(* Logix 5000 project; controller NSH_PLC1 vendor 1 type 14 code 167 rev 32.11; software revision 32.02; part 3 of 12 *)
(* tags used below, declared in another part *)
   M10 : Motor;   // Vib.
   M10A : Motor;   // Asp.
   M10B : Motor;   // Asp.
   M11 : Motor;   // Ele.
   M12aA : Motor;   // Grav.Sep
   M12aB : Motor;   // Syntron
   M13aA : Motor;   // Grav.Sep
   M13aB : Motor;   // Syntron
   M14 : Motor;   // Vib.
   M15 : Motor;   // Ele.
   M1A : Motor;   // Vib.
   M2 : Motor;   // Vib.
   M25 : Motor;   // Accept Vib.
   M27 : Motor;   // Belt
   M28 : Motor;   // Belt
   M29 : Motor;   // Ele.
   M3 : Motor;   // Belt
   M30A : Motor;   // HC Vib.
   M30B : Motor;   // Hard Crkr.
   M30C : Motor;   // Shr.Roll.
   M30D : Motor;   // Shr.Roll.
   M31A : Motor;   // Asp.
   M31B : Motor;   // Asp.
   M32A : Motor;   // Vib.Scrn.
   M32B : Motor;   // Ele.
   M33 : Motor;   // Belt
   M34 : Motor;   // Destoner
   M35 : Motor;   // Ele.
   M36A : Motor;   // G. Sep.
   M36B : Motor;   // R. Feeder.
   M37 : Motor;   // 5x12
   M38A : Motor;   // Asp.
   M38B : Motor;   // Asp.
   M39 : Motor;   // Ele.
   M4 : Motor;   // Vib.
   M40A : Motor;   // Sep.
   M40B : Motor;   // Syn.Fer.
   M41 : Motor;   // Ele.
   M44A : Motor;   // Belt
   M44B : Motor;   // Belt
   M5 : Motor;   // Vib.
   M6 : Motor;   // Belt
   M7 : Motor;   // Ele.
   M8 : Motor;   // Shkr.
   M9A : Motor;   // Asp.
   M9B : Motor;   // Asp.
   S11 : Motor;   // Ele.
   S32A : Motor;   // HC Vib.
   S32B : Motor;   // Hard Crkr.
   S32C : Motor;   // Shr.Roll.
   S32D : Motor;   // S.Roll
   S33A : Motor;   // HC Vib.
   S33B : Motor;   // Hard Crkr.
   S33C : Motor;   // Shr.Roll.
   S33D : Motor;   // S.Roll
   S37A : Motor;   // HC Vib.
   S37B : Motor;   // Hard Crkr.
   S37C : Motor;   // Shr.Roll.
   S37D : Motor;   // S.Roll
   S40A : Motor;   // HC Vib.
   S40B : Motor;   // Hard Crkr.
   S40C : Motor;   // Shr.Roll.
   S40D : Motor;   // S.Roll
   S42A : Motor;   // HC Vib.
   S42B : Motor;   // Hard Crkr.
   S42C : Motor;   // S.Roll
   S42D : Motor;   // Shr.Roll.
   S46A : Motor;   // HC Vib.
   S46B : Motor;   // Hard Crkr.
   S46C : Motor;   // S.Roll
   S46D : Motor;   // Shr.Roll.
(* HullerSheller, continued *)

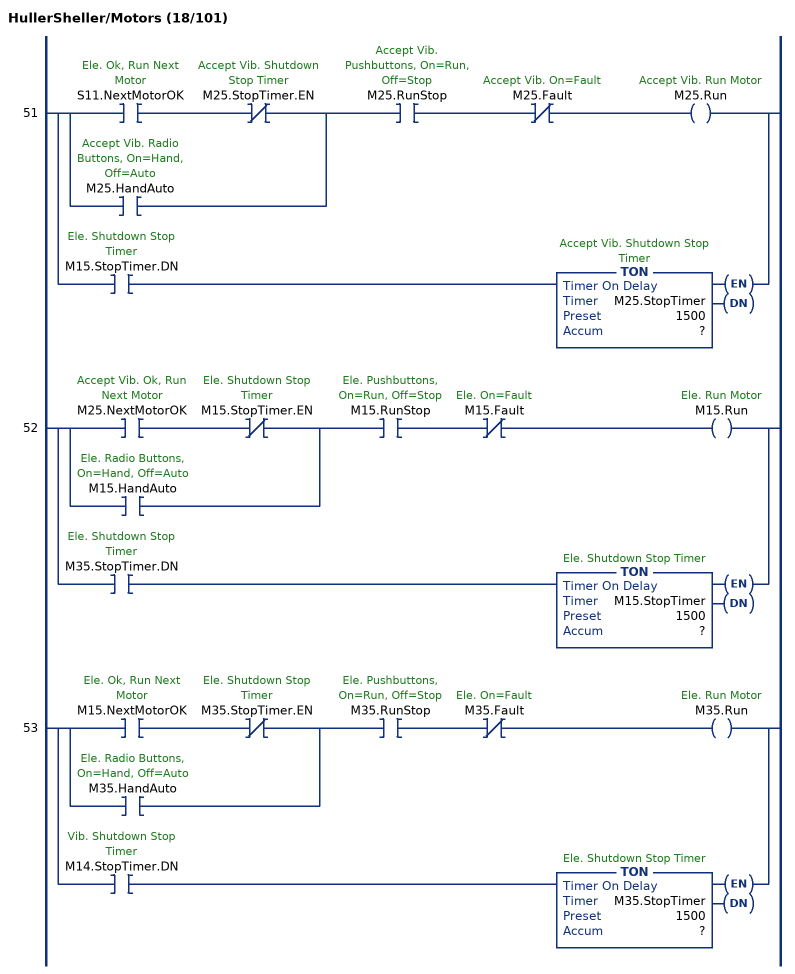
   [picture p42: HullerSheller/Motors rungs 51-53]
   51: [[XIC(S11.NextMotorOK) XIO(M25.StopTimer.EN) ,XIC(M25.HandAuto) ] XIC(M25.RunStop) XIO(M25.Fault) OTE(M25.Run) ,XIC(M15.StopTimer.DN) TON(M25.StopTimer,?,?) ];
   52: [[XIC(M25.NextMotorOK) XIO(M15.StopTimer.EN) ,XIC(M15.HandAuto) ] XIC(M15.RunStop) XIO(M15.Fault) OTE(M15.Run) ,XIC(M35.StopTimer.DN) TON(M15.StopTimer,?,?) ];
   53: [[XIC(M15.NextMotorOK) XIO(M35.StopTimer.EN) ,XIC(M35.HandAuto) ] XIC(M35.RunStop) XIO(M35.Fault) OTE(M35.Run) ,XIC(M14.StopTimer.DN) TON(M35.StopTimer,?,?) ];
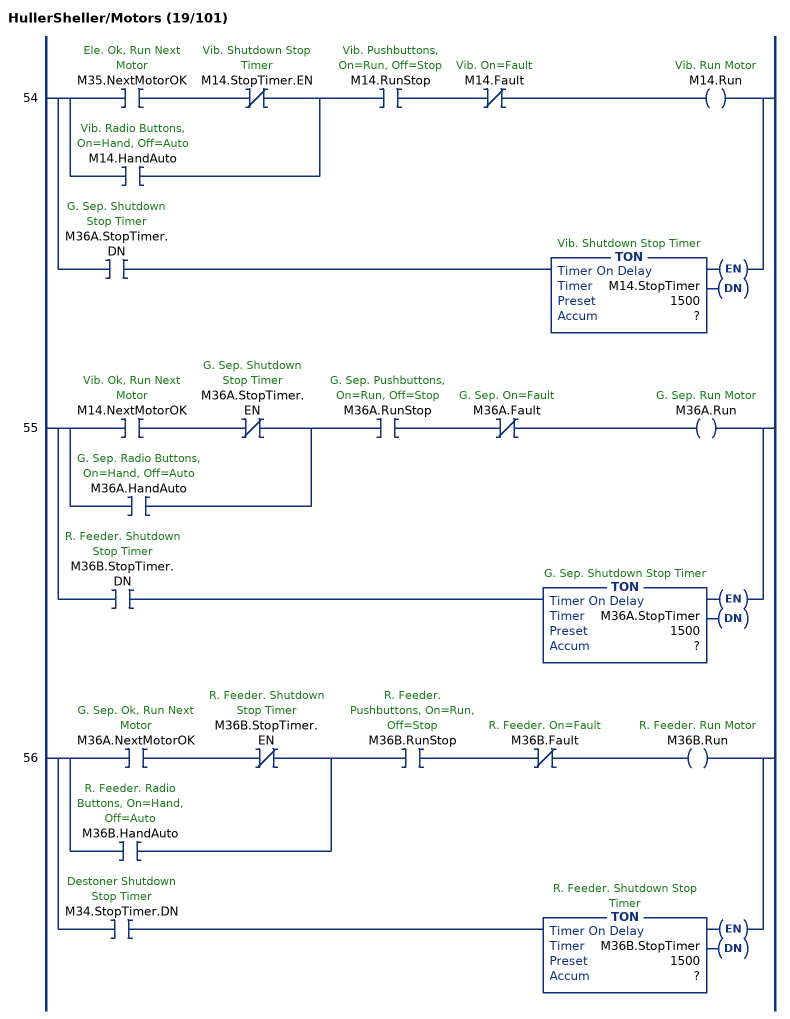
   54: [[XIC(M35.NextMotorOK) XIO(M14.StopTimer.EN) ,XIC(M14.HandAuto) ] XIC(M14.RunStop) XIO(M14.Fault) OTE(M14.Run) ,XIC(M36A.StopTimer.DN) TON(M14.StopTimer,?,?) ];
   55: [[XIC(M14.NextMotorOK) XIO(M36A.StopTimer.EN) ,XIC(M36A.HandAuto) ] XIC(M36A.RunStop) XIO(M36A.Fault) OTE(M36A.Run) ,XIC(M36B.StopTimer.DN) TON(M36A.StopTimer,?,?) ];
   56: [[XIC(M36A.NextMotorOK) XIO(M36B.StopTimer.EN) ,XIC(M36B.HandAuto) ] XIC(M36B.RunStop) XIO(M36B.Fault) OTE(M36B.Run) ,XIC(M34.StopTimer.DN) TON(M36B.StopTimer,?,?) ];
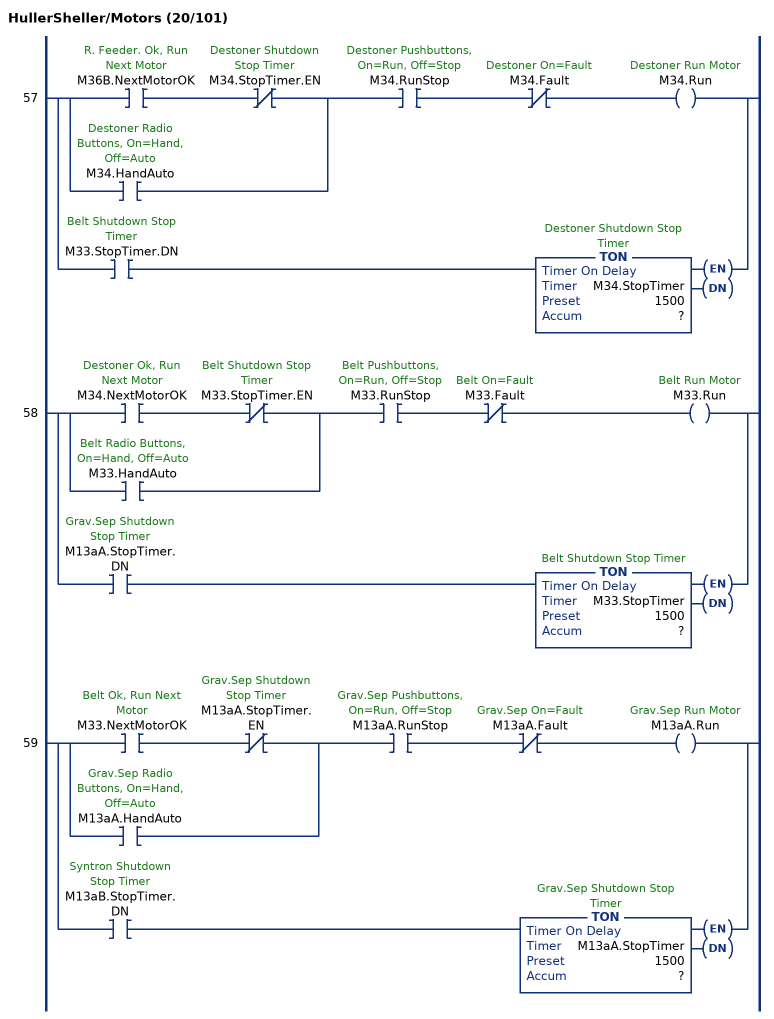
   57: [[XIC(M36B.NextMotorOK) XIO(M34.StopTimer.EN) ,XIC(M34.HandAuto) ] XIC(M34.RunStop) XIO(M34.Fault) OTE(M34.Run) ,XIC(M33.StopTimer.DN) TON(M34.StopTimer,?,?) ];
   58: [[XIC(M34.NextMotorOK) XIO(M33.StopTimer.EN) ,XIC(M33.HandAuto) ] XIC(M33.RunStop) XIO(M33.Fault) OTE(M33.Run) ,XIC(M13aA.StopTimer.DN) TON(M33.StopTimer,?,?) ];
   59: [[XIC(M33.NextMotorOK) XIO(M13aA.StopTimer.EN) ,XIC(M13aA.HandAuto) ] XIC(M13aA.RunStop) XIO(M13aA.Fault) OTE(M13aA.Run) ,XIC(M13aB.StopTimer.DN) TON(M13aA.StopTimer,?,?) ];
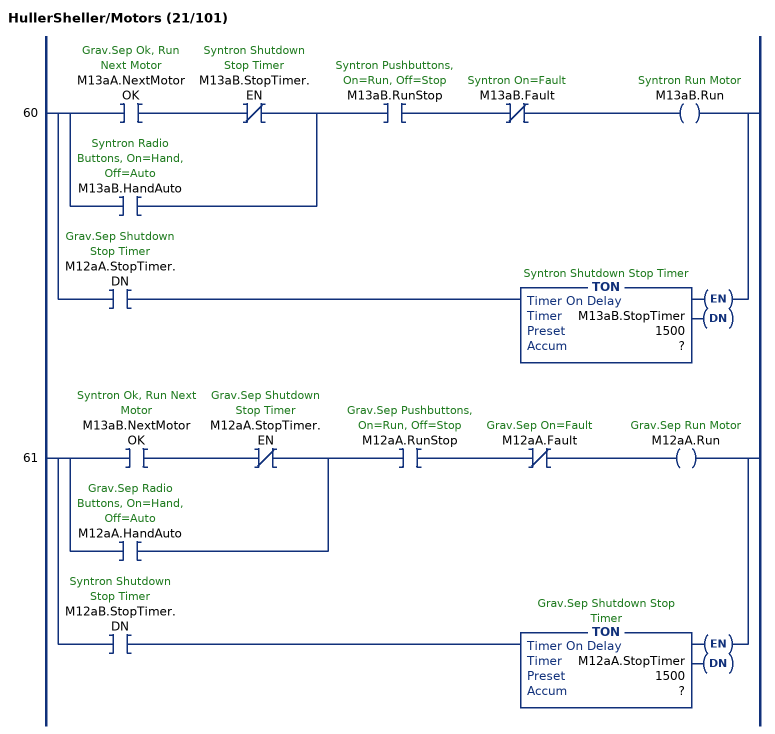
   60: [[XIC(M13aA.NextMotorOK) XIO(M13aB.StopTimer.EN) ,XIC(M13aB.HandAuto) ] XIC(M13aB.RunStop) XIO(M13aB.Fault) OTE(M13aB.Run) ,XIC(M12aA.StopTimer.DN) TON(M13aB.StopTimer,?,?) ];
   61: [[XIC(M13aB.NextMotorOK) XIO(M12aA.StopTimer.EN) ,XIC(M12aA.HandAuto) ] XIC(M12aA.RunStop) XIO(M12aA.Fault) OTE(M12aA.Run) ,XIC(M12aB.StopTimer.DN) TON(M12aA.StopTimer,?,?) ];
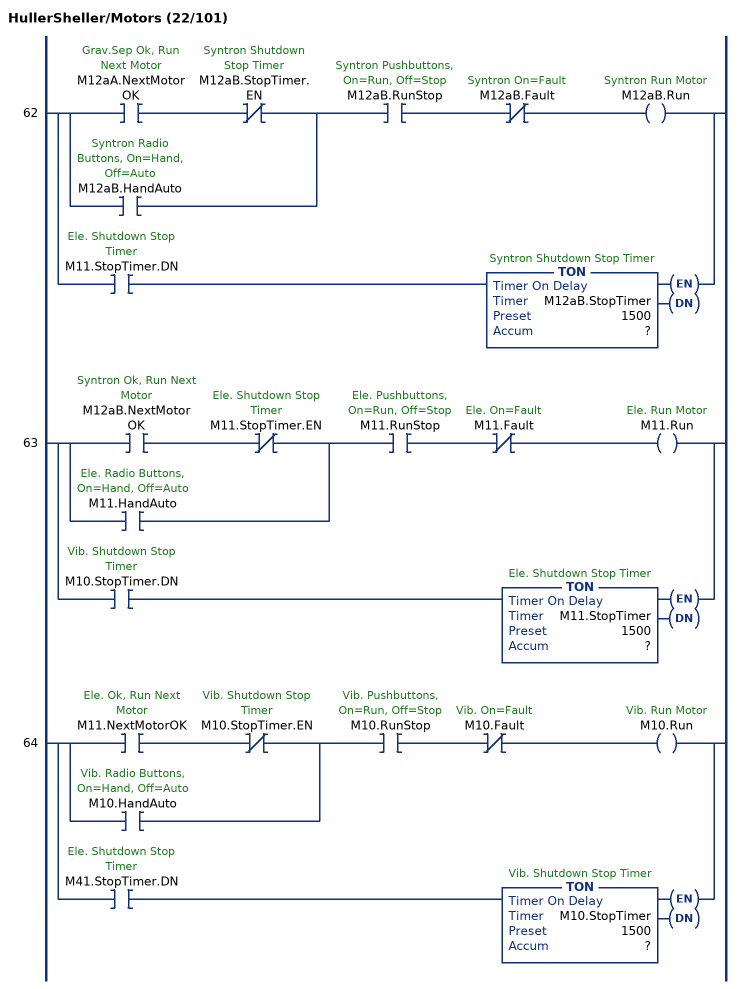
   62: [[XIC(M12aA.NextMotorOK) XIO(M12aB.StopTimer.EN) ,XIC(M12aB.HandAuto) ] XIC(M12aB.RunStop) XIO(M12aB.Fault) OTE(M12aB.Run) ,XIC(M11.StopTimer.DN) TON(M12aB.StopTimer,?,?) ];
   63: [[XIC(M12aB.NextMotorOK) XIO(M11.StopTimer.EN) ,XIC(M11.HandAuto) ] XIC(M11.RunStop) XIO(M11.Fault) OTE(M11.Run) ,XIC(M10.StopTimer.DN) TON(M11.StopTimer,?,?) ];
   64: [[XIC(M11.NextMotorOK) XIO(M10.StopTimer.EN) ,XIC(M10.HandAuto) ] XIC(M10.RunStop) XIO(M10.Fault) OTE(M10.Run) ,XIC(M41.StopTimer.DN) TON(M10.StopTimer,?,?) ];
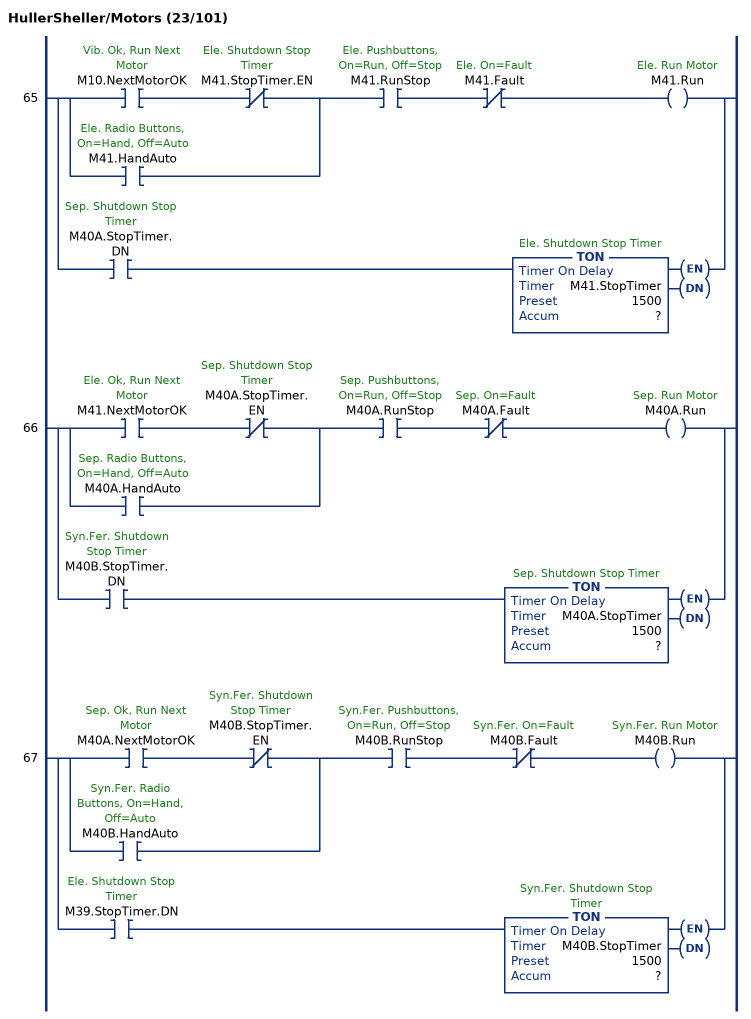
   65: [[XIC(M10.NextMotorOK) XIO(M41.StopTimer.EN) ,XIC(M41.HandAuto) ] XIC(M41.RunStop) XIO(M41.Fault) OTE(M41.Run) ,XIC(M40A.StopTimer.DN) TON(M41.StopTimer,?,?) ];
   66: [[XIC(M41.NextMotorOK) XIO(M40A.StopTimer.EN) ,XIC(M40A.HandAuto) ] XIC(M40A.RunStop) XIO(M40A.Fault) OTE(M40A.Run) ,XIC(M40B.StopTimer.DN) TON(M40A.StopTimer,?,?) ];
   67: [[XIC(M40A.NextMotorOK) XIO(M40B.StopTimer.EN) ,XIC(M40B.HandAuto) ] XIC(M40B.RunStop) XIO(M40B.Fault) OTE(M40B.Run) ,XIC(M39.StopTimer.DN) TON(M40B.StopTimer,?,?) ];
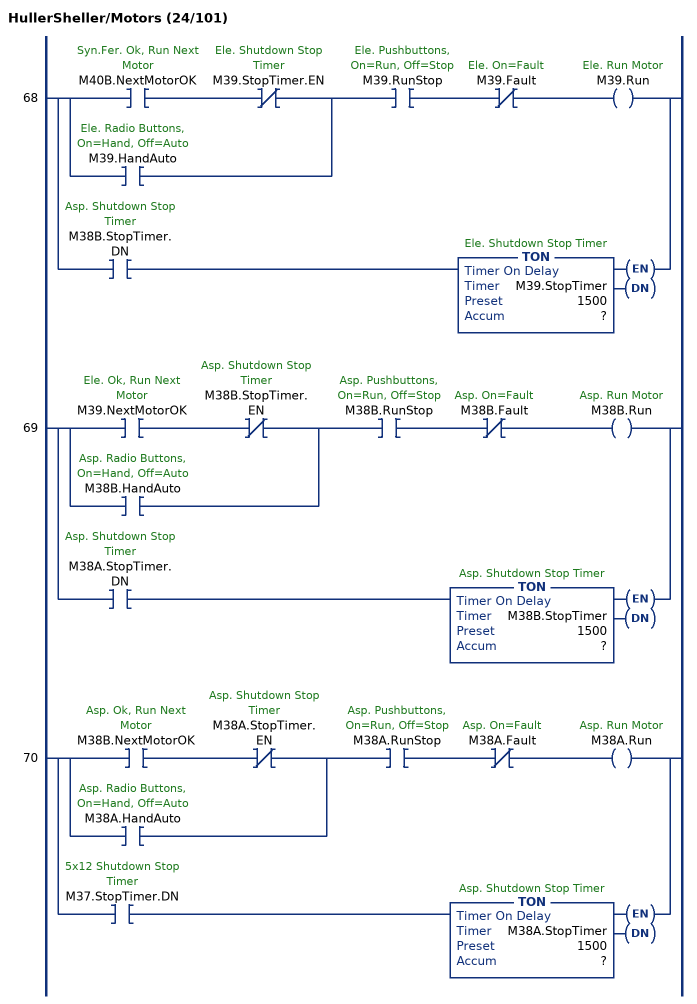
   68: [[XIC(M40B.NextMotorOK) XIO(M39.StopTimer.EN) ,XIC(M39.HandAuto) ] XIC(M39.RunStop) XIO(M39.Fault) OTE(M39.Run) ,XIC(M38B.StopTimer.DN) TON(M39.StopTimer,?,?) ];
   69: [[XIC(M39.NextMotorOK) XIO(M38B.StopTimer.EN) ,XIC(M38B.HandAuto) ] XIC(M38B.RunStop) XIO(M38B.Fault) OTE(M38B.Run) ,XIC(M38A.StopTimer.DN) TON(M38B.StopTimer,?,?) ];
   70: [[XIC(M38B.NextMotorOK) XIO(M38A.StopTimer.EN) ,XIC(M38A.HandAuto) ] XIC(M38A.RunStop) XIO(M38A.Fault) OTE(M38A.Run) ,XIC(M37.StopTimer.DN) TON(M38A.StopTimer,?,?) ];
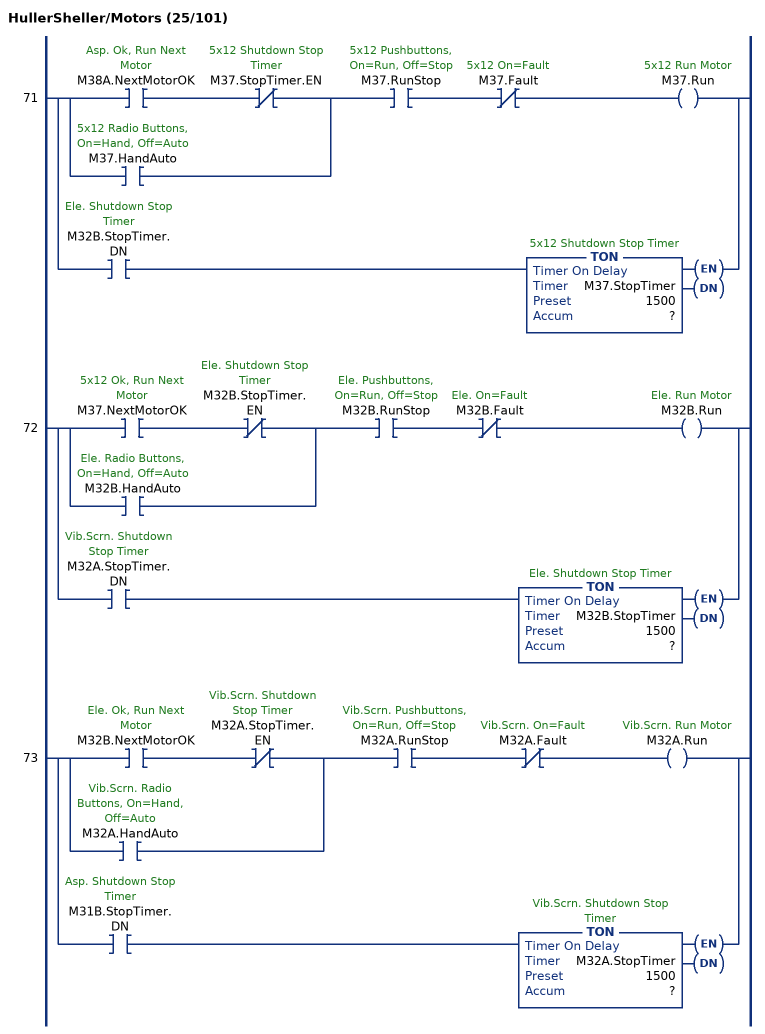
   71: [[XIC(M38A.NextMotorOK) XIO(M37.StopTimer.EN) ,XIC(M37.HandAuto) ] XIC(M37.RunStop) XIO(M37.Fault) OTE(M37.Run) ,XIC(M32B.StopTimer.DN) TON(M37.StopTimer,?,?) ];
   72: [[XIC(M37.NextMotorOK) XIO(M32B.StopTimer.EN) ,XIC(M32B.HandAuto) ] XIC(M32B.RunStop) XIO(M32B.Fault) OTE(M32B.Run) ,XIC(M32A.StopTimer.DN) TON(M32B.StopTimer,?,?) ];
   73: [[XIC(M32B.NextMotorOK) XIO(M32A.StopTimer.EN) ,XIC(M32A.HandAuto) ] XIC(M32A.RunStop) XIO(M32A.Fault) OTE(M32A.Run) ,XIC(M31B.StopTimer.DN) TON(M32A.StopTimer,?,?) ];
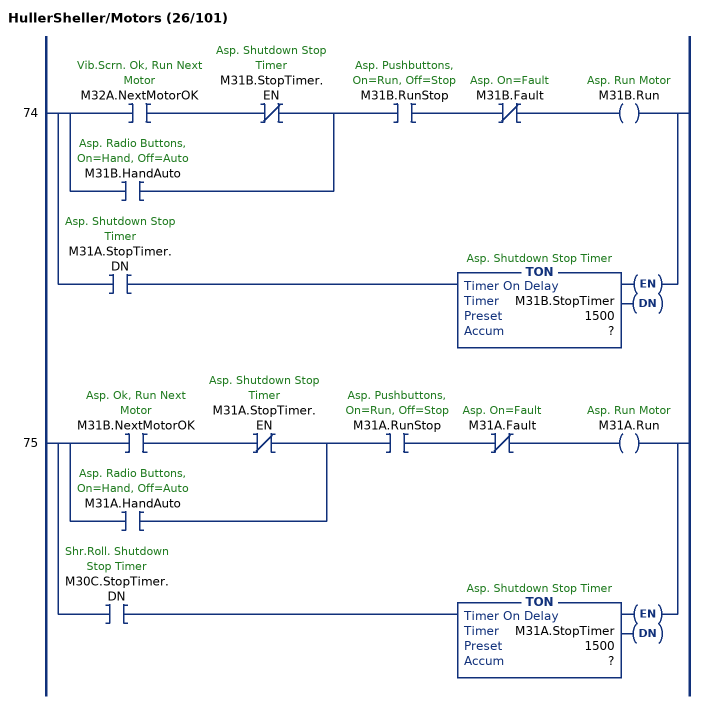
   74: [[XIC(M32A.NextMotorOK) XIO(M31B.StopTimer.EN) ,XIC(M31B.HandAuto) ] XIC(M31B.RunStop) XIO(M31B.Fault) OTE(M31B.Run) ,XIC(M31A.StopTimer.DN) TON(M31B.StopTimer,?,?) ];
   75: [[XIC(M31B.NextMotorOK) XIO(M31A.StopTimer.EN) ,XIC(M31A.HandAuto) ] XIC(M31A.RunStop) XIO(M31A.Fault) OTE(M31A.Run) ,XIC(M30C.StopTimer.DN) TON(M31A.StopTimer,?,?) ];
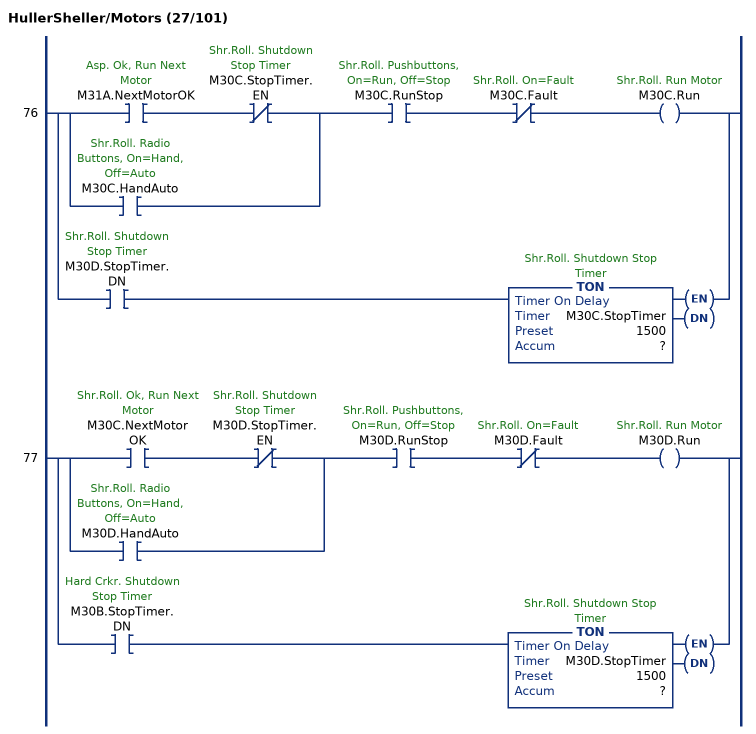
   76: [[XIC(M31A.NextMotorOK) XIO(M30C.StopTimer.EN) ,XIC(M30C.HandAuto) ] XIC(M30C.RunStop) XIO(M30C.Fault) OTE(M30C.Run) ,XIC(M30D.StopTimer.DN) TON(M30C.StopTimer,?,?) ];
   77: [[XIC(M30C.NextMotorOK) XIO(M30D.StopTimer.EN) ,XIC(M30D.HandAuto) ] XIC(M30D.RunStop) XIO(M30D.Fault) OTE(M30D.Run) ,XIC(M30B.StopTimer.DN) TON(M30D.StopTimer,?,?) ];
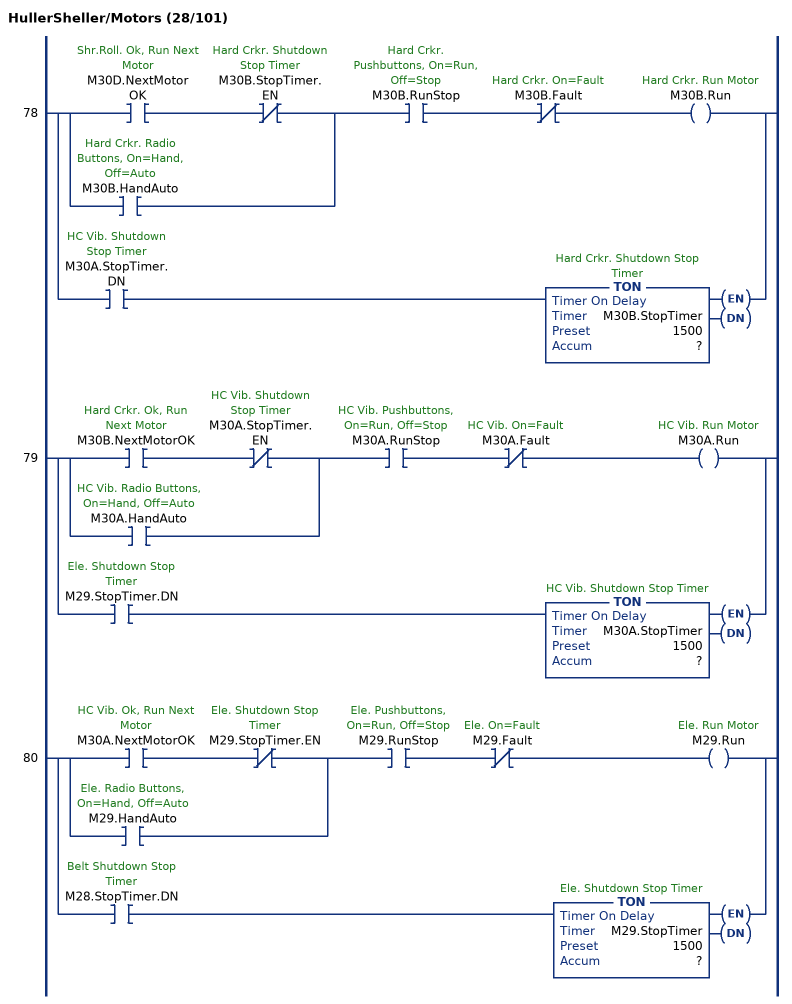
   78: [[XIC(M30D.NextMotorOK) XIO(M30B.StopTimer.EN) ,XIC(M30B.HandAuto) ] XIC(M30B.RunStop) XIO(M30B.Fault) OTE(M30B.Run) ,XIC(M30A.StopTimer.DN) TON(M30B.StopTimer,?,?) ];
   79: [[XIC(M30B.NextMotorOK) XIO(M30A.StopTimer.EN) ,XIC(M30A.HandAuto) ] XIC(M30A.RunStop) XIO(M30A.Fault) OTE(M30A.Run) ,XIC(M29.StopTimer.DN) TON(M30A.StopTimer,?,?) ];
   80: [[XIC(M30A.NextMotorOK) XIO(M29.StopTimer.EN) ,XIC(M29.HandAuto) ] XIC(M29.RunStop) XIO(M29.Fault) OTE(M29.Run) ,XIC(M28.StopTimer.DN) TON(M29.StopTimer,?,?) ];
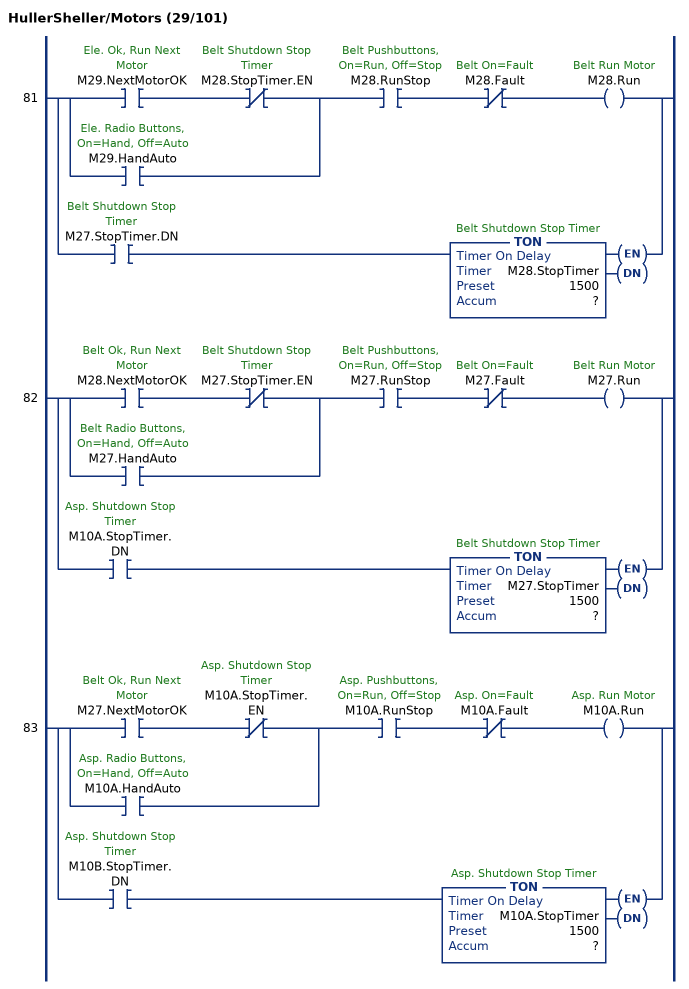
   81: [[XIC(M29.NextMotorOK) XIO(M28.StopTimer.EN) ,XIC(M29.HandAuto) ] XIC(M28.RunStop) XIO(M28.Fault) OTE(M28.Run) ,XIC(M27.StopTimer.DN) TON(M28.StopTimer,?,?) ];
   82: [[XIC(M28.NextMotorOK) XIO(M27.StopTimer.EN) ,XIC(M27.HandAuto) ] XIC(M27.RunStop) XIO(M27.Fault) OTE(M27.Run) ,XIC(M10A.StopTimer.DN) TON(M27.StopTimer,?,?) ];
   83: [[XIC(M27.NextMotorOK) XIO(M10A.StopTimer.EN) ,XIC(M10A.HandAuto) ] XIC(M10A.RunStop) XIO(M10A.Fault) OTE(M10A.Run) ,XIC(M10B.StopTimer.DN) TON(M10A.StopTimer,?,?) ];
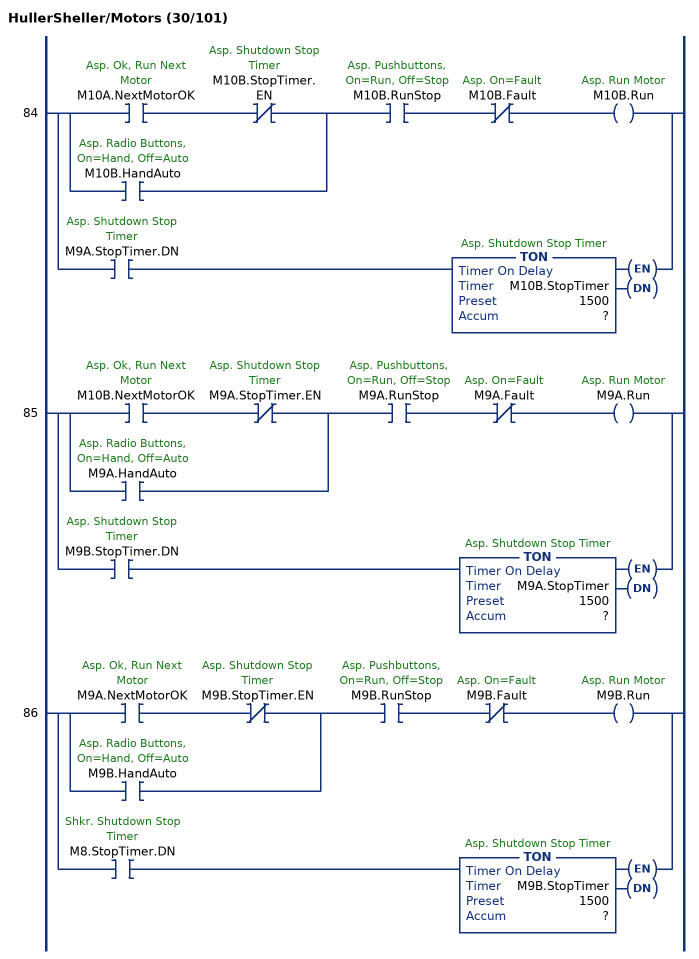
   84: [[XIC(M10A.NextMotorOK) XIO(M10B.StopTimer.EN) ,XIC(M10B.HandAuto) ] XIC(M10B.RunStop) XIO(M10B.Fault) OTE(M10B.Run) ,XIC(M9A.StopTimer.DN) TON(M10B.StopTimer,?,?) ];
   85: [[XIC(M10B.NextMotorOK) XIO(M9A.StopTimer.EN) ,XIC(M9A.HandAuto) ] XIC(M9A.RunStop) XIO(M9A.Fault) OTE(M9A.Run) ,XIC(M9B.StopTimer.DN) TON(M9A.StopTimer,?,?) ];
   86: [[XIC(M9A.NextMotorOK) XIO(M9B.StopTimer.EN) ,XIC(M9B.HandAuto) ] XIC(M9B.RunStop) XIO(M9B.Fault) OTE(M9B.Run) ,XIC(M8.StopTimer.DN) TON(M9B.StopTimer,?,?) ];
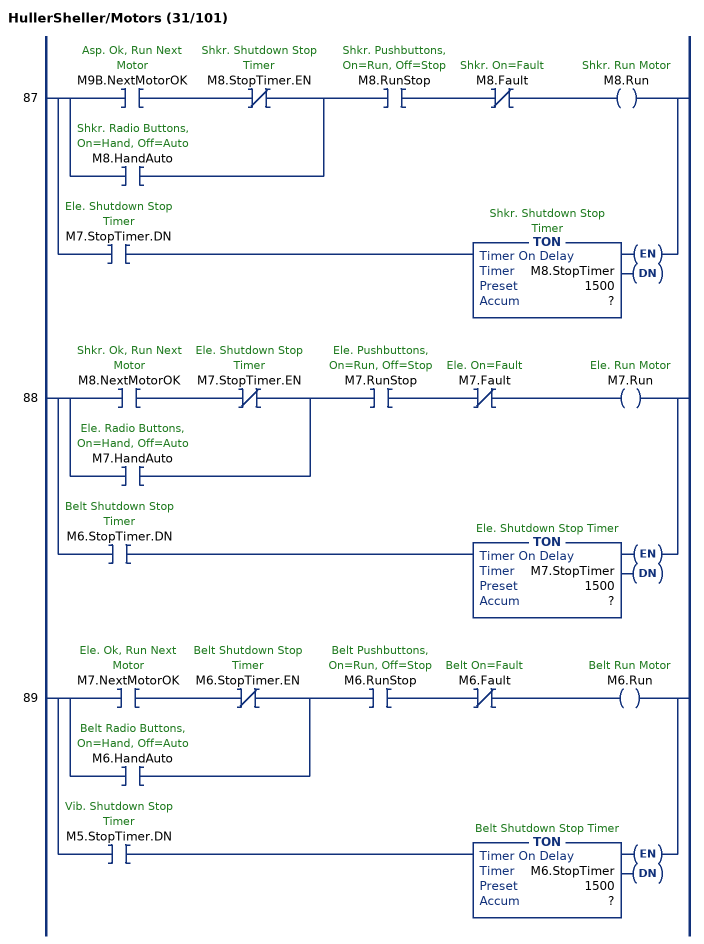
   87: [[XIC(M9B.NextMotorOK) XIO(M8.StopTimer.EN) ,XIC(M8.HandAuto) ] XIC(M8.RunStop) XIO(M8.Fault) OTE(M8.Run) ,XIC(M7.StopTimer.DN) TON(M8.StopTimer,?,?) ];
   88: [[XIC(M8.NextMotorOK) XIO(M7.StopTimer.EN) ,XIC(M7.HandAuto) ] XIC(M7.RunStop) XIO(M7.Fault) OTE(M7.Run) ,XIC(M6.StopTimer.DN) TON(M7.StopTimer,?,?) ];
   89: [[XIC(M7.NextMotorOK) XIO(M6.StopTimer.EN) ,XIC(M6.HandAuto) ] XIC(M6.RunStop) XIO(M6.Fault) OTE(M6.Run) ,XIC(M5.StopTimer.DN) TON(M6.StopTimer,?,?) ];
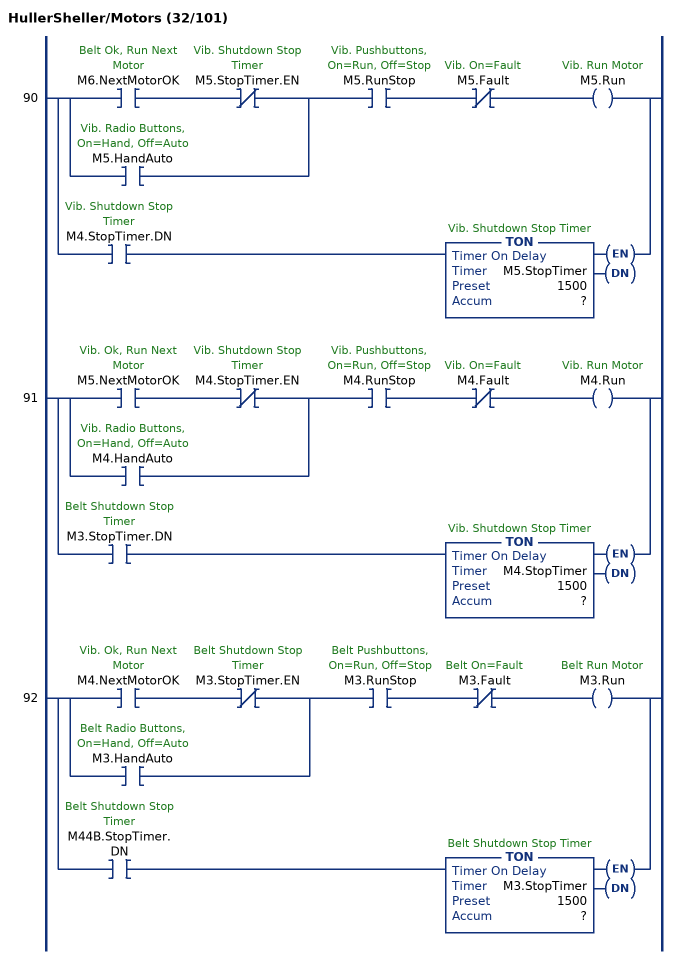
   90: [[XIC(M6.NextMotorOK) XIO(M5.StopTimer.EN) ,XIC(M5.HandAuto) ] XIC(M5.RunStop) XIO(M5.Fault) OTE(M5.Run) ,XIC(M4.StopTimer.DN) TON(M5.StopTimer,?,?) ];
   91: [[XIC(M5.NextMotorOK) XIO(M4.StopTimer.EN) ,XIC(M4.HandAuto) ] XIC(M4.RunStop) XIO(M4.Fault) OTE(M4.Run) ,XIC(M3.StopTimer.DN) TON(M4.StopTimer,?,?) ];
   92: [[XIC(M4.NextMotorOK) XIO(M3.StopTimer.EN) ,XIC(M3.HandAuto) ] XIC(M3.RunStop) XIO(M3.Fault) OTE(M3.Run) ,XIC(M44B.StopTimer.DN) TON(M3.StopTimer,?,?) ];
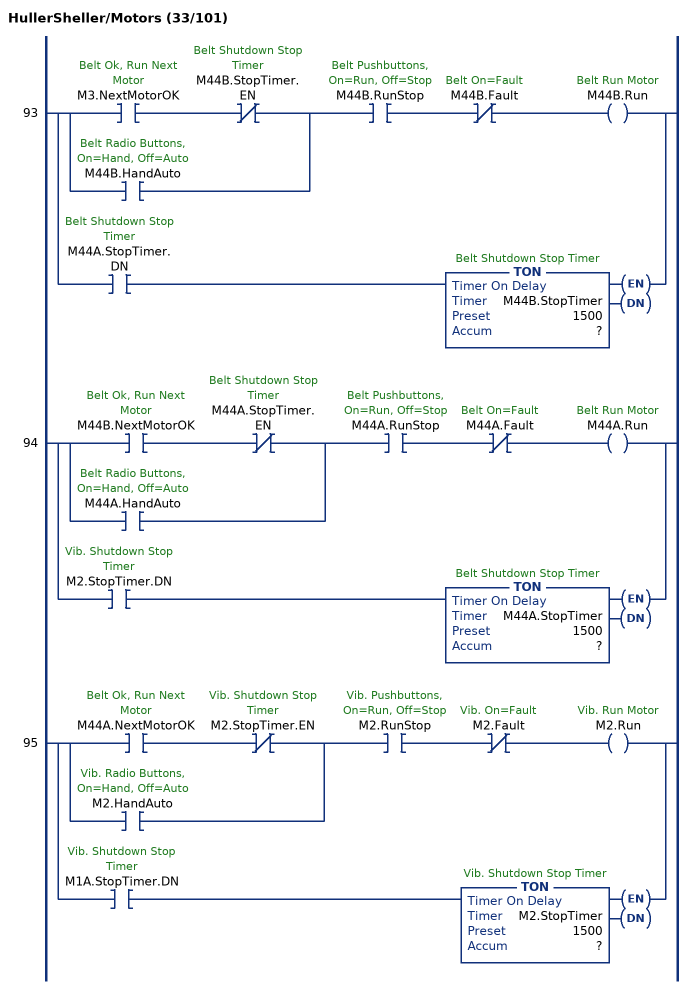
   93: [[XIC(M3.NextMotorOK) XIO(M44B.StopTimer.EN) ,XIC(M44B.HandAuto) ] XIC(M44B.RunStop) XIO(M44B.Fault) OTE(M44B.Run) ,XIC(M44A.StopTimer.DN) TON(M44B.StopTimer,?,?) ];
   94: [[XIC(M44B.NextMotorOK) XIO(M44A.StopTimer.EN) ,XIC(M44A.HandAuto) ] XIC(M44A.RunStop) XIO(M44A.Fault) OTE(M44A.Run) ,XIC(M2.StopTimer.DN) TON(M44A.StopTimer,?,?) ];
   95: [[XIC(M44A.NextMotorOK) XIO(M2.StopTimer.EN) ,XIC(M2.HandAuto) ] XIC(M2.RunStop) XIO(M2.Fault) OTE(M2.Run) ,XIC(M1A.StopTimer.DN) TON(M2.StopTimer,?,?) ];
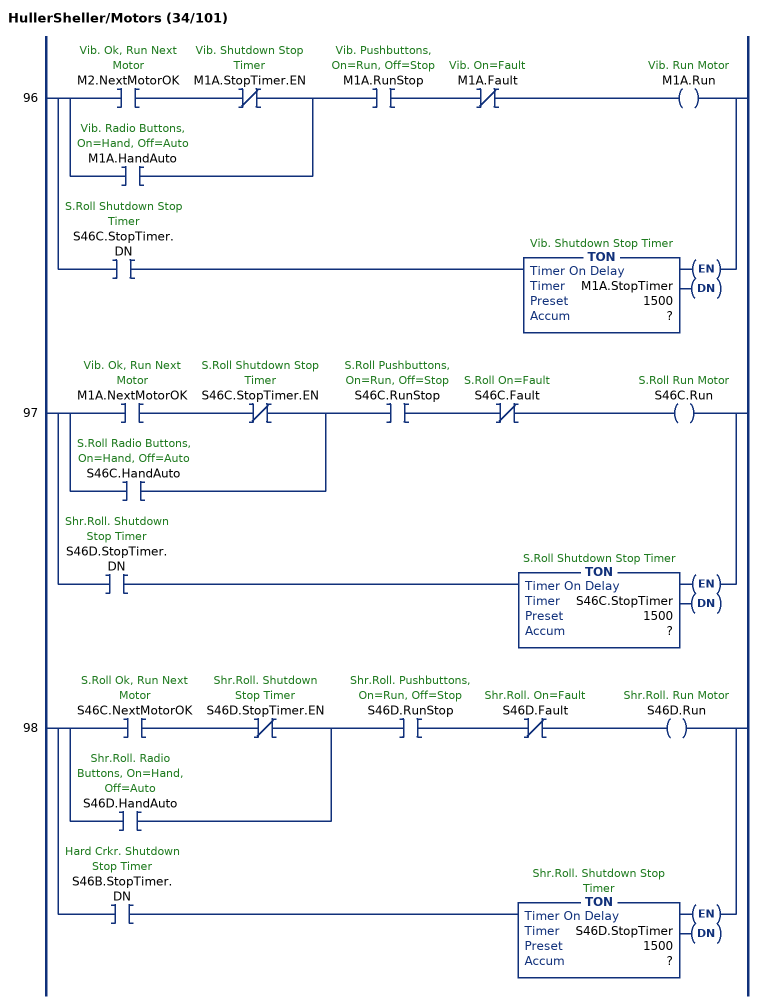
   96: [[XIC(M2.NextMotorOK) XIO(M1A.StopTimer.EN) ,XIC(M1A.HandAuto) ] XIC(M1A.RunStop) XIO(M1A.Fault) OTE(M1A.Run) ,XIC(S46C.StopTimer.DN) TON(M1A.StopTimer,?,?) ];
   97: [[XIC(M1A.NextMotorOK) XIO(S46C.StopTimer.EN) ,XIC(S46C.HandAuto) ] XIC(S46C.RunStop) XIO(S46C.Fault) OTE(S46C.Run) ,XIC(S46D.StopTimer.DN) TON(S46C.StopTimer,?,?) ];
   98: [[XIC(S46C.NextMotorOK) XIO(S46D.StopTimer.EN) ,XIC(S46D.HandAuto) ] XIC(S46D.RunStop) XIO(S46D.Fault) OTE(S46D.Run) ,XIC(S46B.StopTimer.DN) TON(S46D.StopTimer,?,?) ];
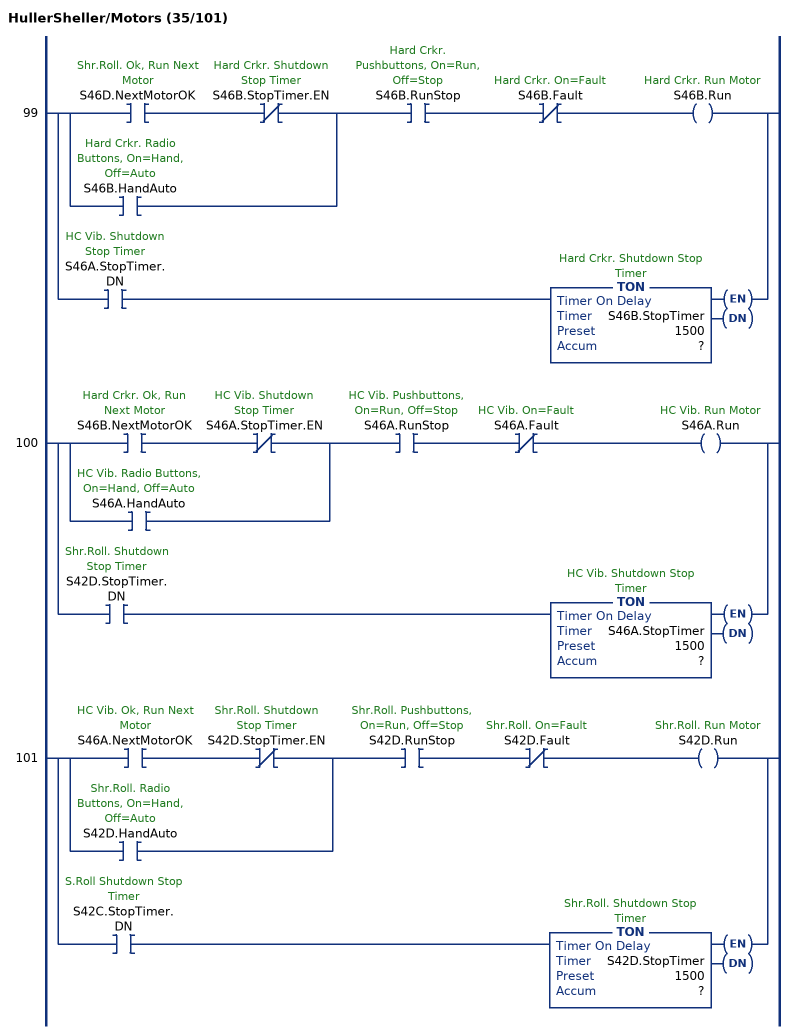
   99: [[XIC(S46D.NextMotorOK) XIO(S46B.StopTimer.EN) ,XIC(S46B.HandAuto) ] XIC(S46B.RunStop) XIO(S46B.Fault) OTE(S46B.Run) ,XIC(S46A.StopTimer.DN) TON(S46B.StopTimer,?,?) ];
   100: [[XIC(S46B.NextMotorOK) XIO(S46A.StopTimer.EN) ,XIC(S46A.HandAuto) ] XIC(S46A.RunStop) XIO(S46A.Fault) OTE(S46A.Run) ,XIC(S42D.StopTimer.DN) TON(S46A.StopTimer,?,?) ];
   101: [[XIC(S46A.NextMotorOK) XIO(S42D.StopTimer.EN) ,XIC(S42D.HandAuto) ] XIC(S42D.RunStop) XIO(S42D.Fault) OTE(S42D.Run) ,XIC(S42C.StopTimer.DN) TON(S42D.StopTimer,?,?) ];
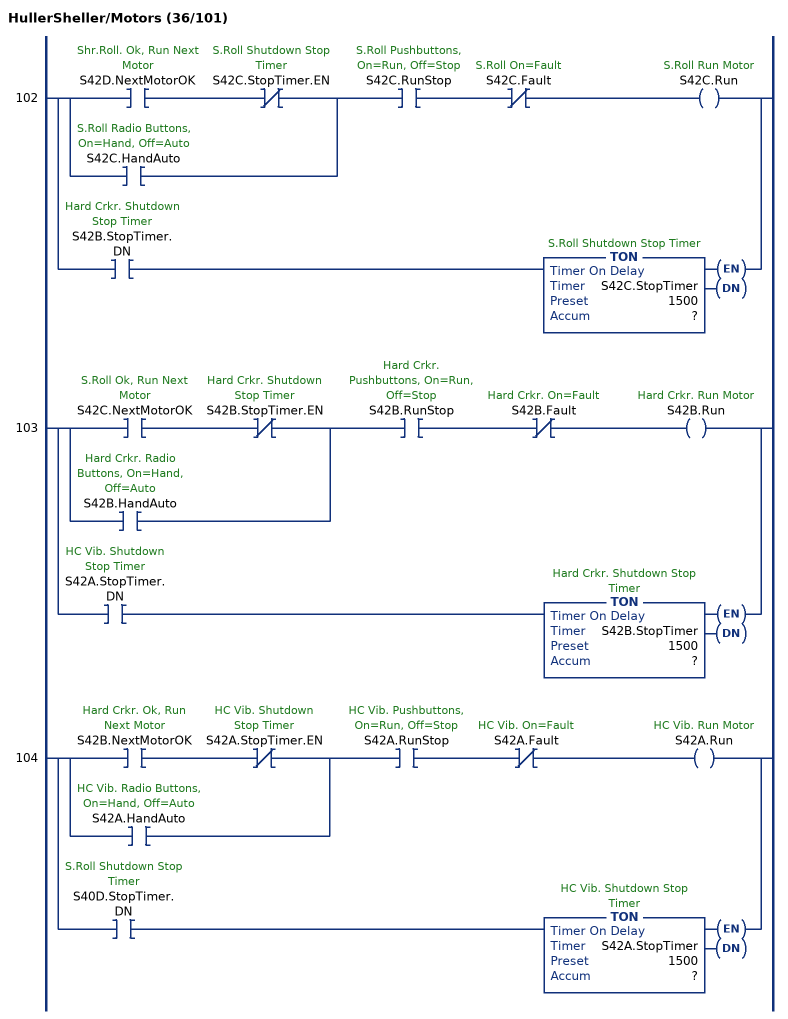
   102: [[XIC(S42D.NextMotorOK) XIO(S42C.StopTimer.EN) ,XIC(S42C.HandAuto) ] XIC(S42C.RunStop) XIO(S42C.Fault) OTE(S42C.Run) ,XIC(S42B.StopTimer.DN) TON(S42C.StopTimer,?,?) ];
   103: [[XIC(S42C.NextMotorOK) XIO(S42B.StopTimer.EN) ,XIC(S42B.HandAuto) ] XIC(S42B.RunStop) XIO(S42B.Fault) OTE(S42B.Run) ,XIC(S42A.StopTimer.DN) TON(S42B.StopTimer,?,?) ];
   104: [[XIC(S42B.NextMotorOK) XIO(S42A.StopTimer.EN) ,XIC(S42A.HandAuto) ] XIC(S42A.RunStop) XIO(S42A.Fault) OTE(S42A.Run) ,XIC(S40D.StopTimer.DN) TON(S42A.StopTimer,?,?) ];
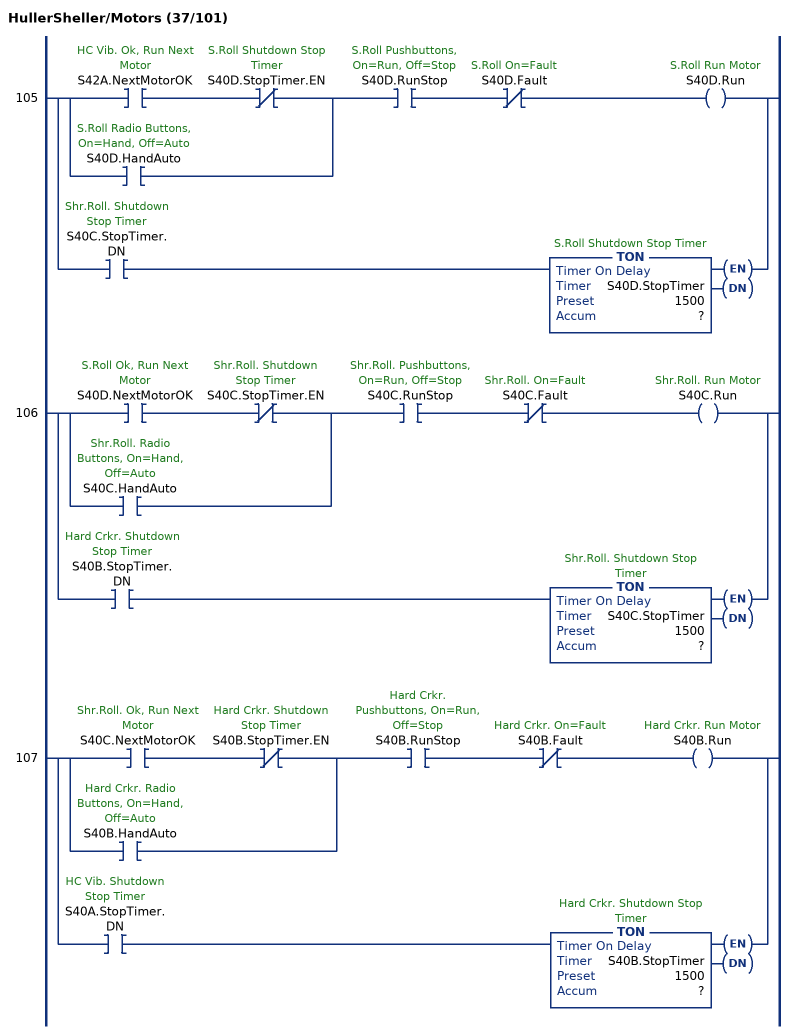
   105: [[XIC(S42A.NextMotorOK) XIO(S40D.StopTimer.EN) ,XIC(S40D.HandAuto) ] XIC(S40D.RunStop) XIO(S40D.Fault) OTE(S40D.Run) ,XIC(S40C.StopTimer.DN) TON(S40D.StopTimer,?,?) ];
   106: [[XIC(S40D.NextMotorOK) XIO(S40C.StopTimer.EN) ,XIC(S40C.HandAuto) ] XIC(S40C.RunStop) XIO(S40C.Fault) OTE(S40C.Run) ,XIC(S40B.StopTimer.DN) TON(S40C.StopTimer,?,?) ];
   107: [[XIC(S40C.NextMotorOK) XIO(S40B.StopTimer.EN) ,XIC(S40B.HandAuto) ] XIC(S40B.RunStop) XIO(S40B.Fault) OTE(S40B.Run) ,XIC(S40A.StopTimer.DN) TON(S40B.StopTimer,?,?) ];
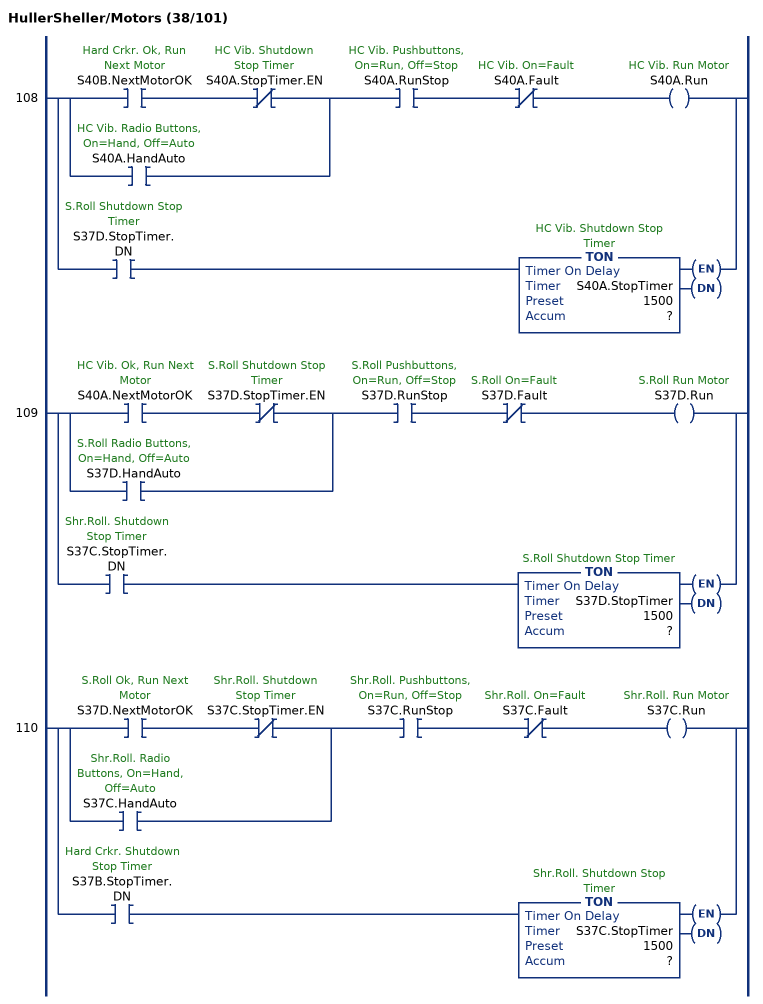
   108: [[XIC(S40B.NextMotorOK) XIO(S40A.StopTimer.EN) ,XIC(S40A.HandAuto) ] XIC(S40A.RunStop) XIO(S40A.Fault) OTE(S40A.Run) ,XIC(S37D.StopTimer.DN) TON(S40A.StopTimer,?,?) ];
   109: [[XIC(S40A.NextMotorOK) XIO(S37D.StopTimer.EN) ,XIC(S37D.HandAuto) ] XIC(S37D.RunStop) XIO(S37D.Fault) OTE(S37D.Run) ,XIC(S37C.StopTimer.DN) TON(S37D.StopTimer,?,?) ];
   110: [[XIC(S37D.NextMotorOK) XIO(S37C.StopTimer.EN) ,XIC(S37C.HandAuto) ] XIC(S37C.RunStop) XIO(S37C.Fault) OTE(S37C.Run) ,XIC(S37B.StopTimer.DN) TON(S37C.StopTimer,?,?) ];
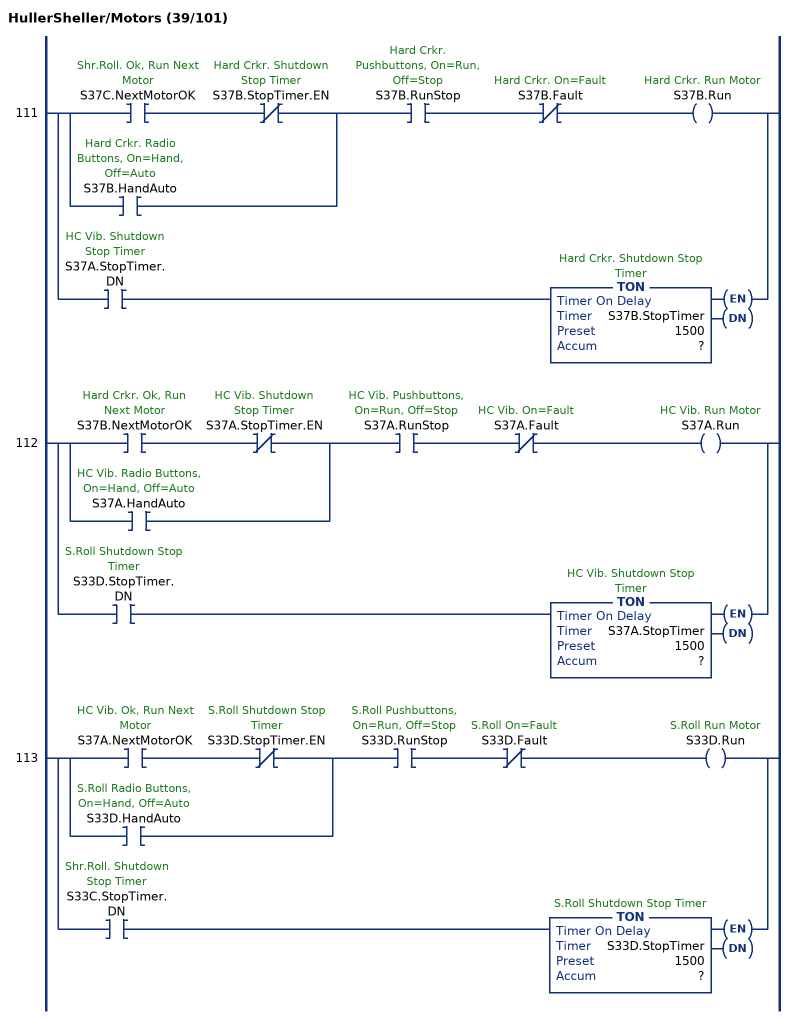
   111: [[XIC(S37C.NextMotorOK) XIO(S37B.StopTimer.EN) ,XIC(S37B.HandAuto) ] XIC(S37B.RunStop) XIO(S37B.Fault) OTE(S37B.Run) ,XIC(S37A.StopTimer.DN) TON(S37B.StopTimer,?,?) ];
   112: [[XIC(S37B.NextMotorOK) XIO(S37A.StopTimer.EN) ,XIC(S37A.HandAuto) ] XIC(S37A.RunStop) XIO(S37A.Fault) OTE(S37A.Run) ,XIC(S33D.StopTimer.DN) TON(S37A.StopTimer,?,?) ];
   113: [[XIC(S37A.NextMotorOK) XIO(S33D.StopTimer.EN) ,XIC(S33D.HandAuto) ] XIC(S33D.RunStop) XIO(S33D.Fault) OTE(S33D.Run) ,XIC(S33C.StopTimer.DN) TON(S33D.StopTimer,?,?) ];
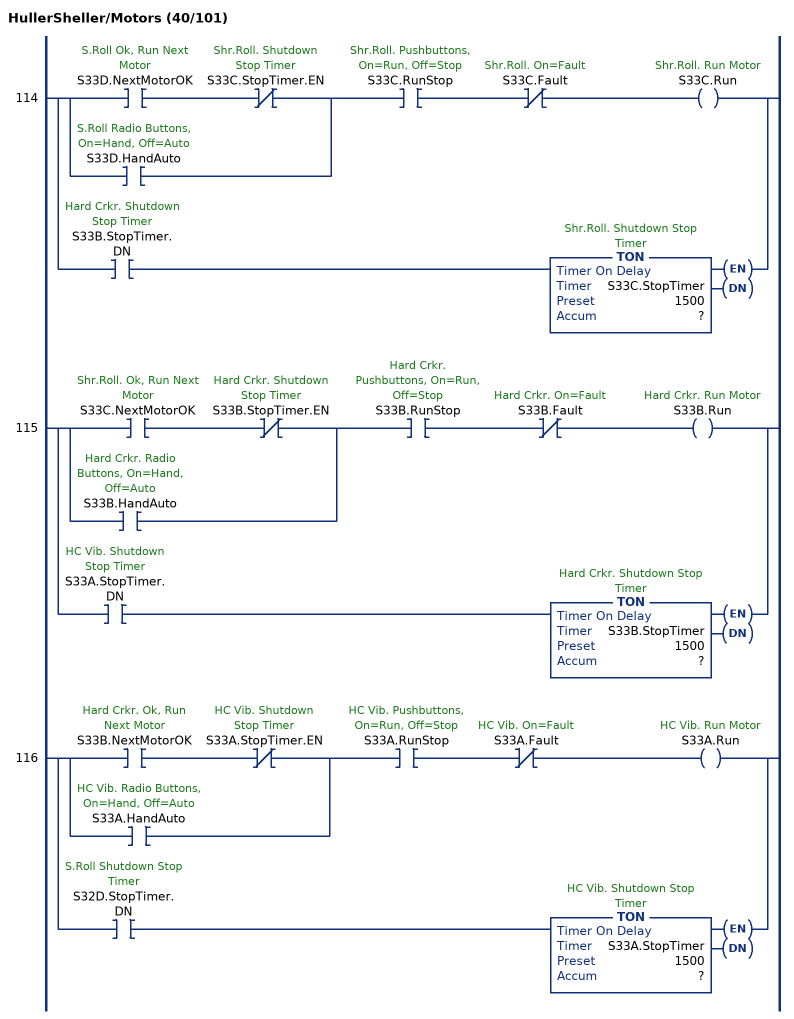
   114: [[XIC(S33D.NextMotorOK) XIO(S33C.StopTimer.EN) ,XIC(S33D.HandAuto) ] XIC(S33C.RunStop) XIO(S33C.Fault) OTE(S33C.Run) ,XIC(S33B.StopTimer.DN) TON(S33C.StopTimer,?,?) ];
   115: [[XIC(S33C.NextMotorOK) XIO(S33B.StopTimer.EN) ,XIC(S33B.HandAuto) ] XIC(S33B.RunStop) XIO(S33B.Fault) OTE(S33B.Run) ,XIC(S33A.StopTimer.DN) TON(S33B.StopTimer,?,?) ];
   116: [[XIC(S33B.NextMotorOK) XIO(S33A.StopTimer.EN) ,XIC(S33A.HandAuto) ] XIC(S33A.RunStop) XIO(S33A.Fault) OTE(S33A.Run) ,XIC(S32D.StopTimer.DN) TON(S33A.StopTimer,?,?) ];
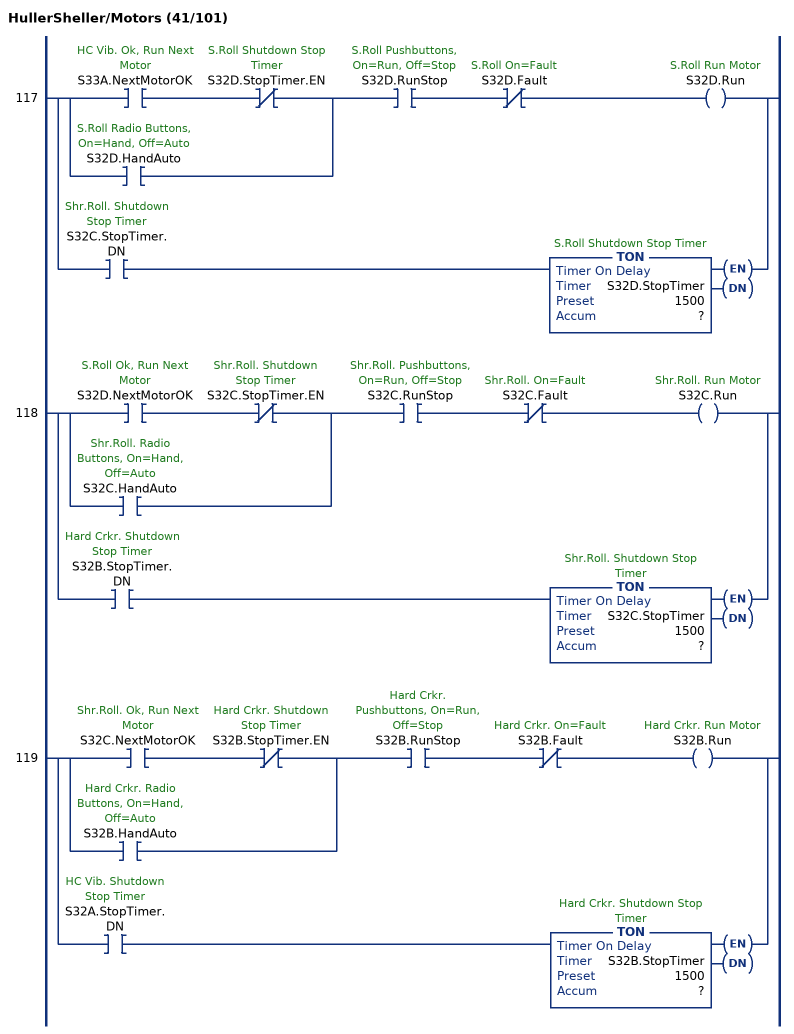
   117: [[XIC(S33A.NextMotorOK) XIO(S32D.StopTimer.EN) ,XIC(S32D.HandAuto) ] XIC(S32D.RunStop) XIO(S32D.Fault) OTE(S32D.Run) ,XIC(S32C.StopTimer.DN) TON(S32D.StopTimer,?,?) ];
   118: [[XIC(S32D.NextMotorOK) XIO(S32C.StopTimer.EN) ,XIC(S32C.HandAuto) ] XIC(S32C.RunStop) XIO(S32C.Fault) OTE(S32C.Run) ,XIC(S32B.StopTimer.DN) TON(S32C.StopTimer,?,?) ];
   119: [[XIC(S32C.NextMotorOK) XIO(S32B.StopTimer.EN) ,XIC(S32B.HandAuto) ] XIC(S32B.RunStop) XIO(S32B.Fault) OTE(S32B.Run) ,XIC(S32A.StopTimer.DN) TON(S32B.StopTimer,?,?) ];
